{attribute 'linkalways'} 
{attribute 'no_explicit_call' := 'This FB is a CLASS and must be accessed using methods or properties'}
{attribute 'enable_dynamic_creation'}
FUNCTION_BLOCK Node_F_VN_MinElementElementwise_TcVnPoint2_DINT EXTENDS VisionNode
VAR
    ipContainer : _ITcVnContainer;
    aMin : _TcVnPoint2_DINT;
    hrPrev : _HRESULT(S_OK);
    hresult : _HRESULT(S_OK);
END_VAR

METHOD PUBLIC  Clone : I_Node
VAR
	pNode : POINTER TO Node_F_VN_MinElementElementwise_TcVnPoint2_DINT;
END_VAR
pNode := __NEW(Node_F_VN_MinElementElementwise_TcVnPoint2_DINT);
Clone := pNode^;
END_METHOD

METHOD FB_init : BOOL
VAR_INPUT
	bInitRetains : BOOL; // if TRUE, the retain variables are initialized (warm start / cold start)
	bInCopyCode : BOOL;  // if TRUE, the instance afterwards gets moved into the copy code (online change)
END_VAR
AddInput('ipContainer', ipContainer);
AddInput('aMin', aMin);
AddInput('hrPrev', hrPrev);
AddOutput('ipContainer', ipContainer);
AddOutput('hresult',hresult);
END_METHOD

METHOD PROTECTED OnExecute : HRESULT
hresult.Value := F_VN_MinElementElementwise_TcVnPoint2_DINT(
    ipContainer := ipContainer.Value,
    aMin := aMin.Value,
    hrPrev:= hrPrev.Value);
END_METHOD

METHOD PUBLIC PreExecutionCheck
VAR_INPUT
	Check : I_PreExecutionChecks;
END_VAR
Check.IsTrue(ipContainer.IsValid, 'ipContainer must be a valid container');
END_METHOD

END_FUNCTION_BLOCK

(* stored: Version 1.1.0.1, ProductVersion 3.1.4024.13
   POU Node_F_VN_MinElementElementwise_TcVnPoint2_DINT: Id {ff4f0d71-503e-4333-ac72-267ec1441a12}, SpecialFunc None
   Folder Constructor: Id {b01b7e6d-1436-41a1-ac5b-66c4945fe505}
   Method Clone: Id {9324e282-f857-4060-8e03-7b73b7aac7af}
   Method FB_init: Id {2cce0a31-fa5b-4ae3-b32b-7aedf10bae40}
   Method OnExecute: Id {665dae8f-a5c4-452b-a583-dcbb688cc263}
   Method PreExecutionCheck: Id {0f82ef59-e913-44ca-af9b-b37fc8324e95} *)
